{attribute 'GeneratedUsingTerminal: EK1100-0000-0018'}
{attribute addProperty BoxType "EK1100-0000-0018"}
{attribute addProperty Id "Beckhoff_EJ5xxxEK1122Beckhoff_EJ5xxxEK1122_A82C313A2A_0001_EJ5002_0000_0016EJ5002_0A956A2724A_0002_EJ5002_0000_0017EJ5002_3C07B65526A_0003_EJ5101_0000_0016EJ5101_D1B6078A30A_0004_EJ5151_0000_0016EJ5151_E1861F5128"}
{attribute addProperty CRC "891182372"}
{attribute addProperty Size "110"}
TYPE Beckhoff_EJ5xxx_351E5D24 EXTENDS EK1100_1FC0878B :
STRUCT
	{attribute addProperty Name "Beckhoff_EJ5xxxEK1122"}
	{attribute addProperty PreviousPort "Beckhoff EJ5xxx : B"}
	Beckhoff_EJ5xxxEK1122 : Beckhoff_EJ5xxxEK1122_A82C313A;
	{attribute addProperty Name "A_0001_EJ5002_0000_0016"}
	{attribute addProperty PreviousPort "Beckhoff EJ5xxxEK1122 : C"}
	A_0001_EJ5002_0000_0016 : EJ5002_0A956A27;
	{attribute addProperty Name "A_0002_EJ5002_0000_0017"}
	{attribute addProperty PreviousPort "A_0001(EJ5002-0000-0016) : B"}
	A_0002_EJ5002_0000_0017 : EJ5002_3C07B655;
	{attribute addProperty Name "A_0003_EJ5101_0000_0016"}
	{attribute addProperty PreviousPort "A_0002(EJ5002-0000-0017) : B"}
	A_0003_EJ5101_0000_0016 : EJ5101_D1B6078A;
	{attribute addProperty Name "A_0004_EJ5151_0000_0016"}
	{attribute addProperty PreviousPort "A_0003(EJ5101-0000-0016) : B"}
	A_0004_EJ5151_0000_0016 : EJ5151_E1861F51;
END_STRUCT
END_TYPE

(* stored: Version 1.2.0.0, ProductVersion 3.1.4024.9
   DUT Beckhoff_EJ5xxx_351E5D24: Id {90866532-405a-48ea-a5ab-d5fdca9f158e} *)
